// TwinCAT 3 PLC project virtual_plc
// ProgramVersion: 3.1.4024.0
// libraries:
//   Tc2_Standard, * (Beckhoff Automation GmbH)
//   Tc2_System, * (Beckhoff Automation GmbH)
//   Tc3_Module, * (Beckhoff Automation GmbH)
//   VisuSymbols,3.5.10.0,System
// project tree:
//   / Gestore di visualizzazione.TcVMO (not stored), GlobalTextList.TcGTLO, PlcTask.TcTTO
//   GVLs/ GVL.TcGVL
//   POUs/ LogMessage.TcPOU, MAIN.TcPOU, MaintenanceTask.TcPOU, status.TcDUT
//   VISU/ Visualization.TcVIS
// real-time tasks:
//   TASK PlcTask: cycle T#10ms, priority 20, ADS port 350

CONFIGURATION virtual_plc
    RESOURCE PLC ON TwinCAT3
        TASK PlcTask(INTERVAL := T#10ms, PRIORITY := 20);
        PROGRAM MAIN WITH PlcTask : MAIN;
    END_RESOURCE
END_CONFIGURATION

// ---- POUs/status.TcDUT
{attribute 'qualified_only'}
{attribute 'strict'}
TYPE status :
(START,
LEVELCHECK,
FILL,
HEAT,
HEATING,
BREW,
WATERREADY,
INTENSITY,
SUGAR,
READY,
CLEAN,
END,
OldState
) := START;
END_TYPE

// ---- GVLs/GVL.TcGVL
{attribute 'qualified_only'}
VAR_GLOBAL
	CoffeeReady: BOOL := FALSE;

	CLEANING: BOOL := FALSE;

	Message: STRING;
END_VAR

// ---- POUs/MAIN.TcPOU
PROGRAM MAIN

VAR
	start : BOOL := FALSE;
	Tfill: TON;
	FILLING : BOOL := FALSE;
	WaterLevel : BOOL := FALSE;
	Level : REAL;
	Theat: TON;
    WaterTemp :REAL;
	HEATING : BOOL := FALSE;
	Tbrew: TON;
    WaterReady : BOOL := FALSE;
	BREWING : BOOL := FALSE;
    Tend: TON;
	
	CoffeeBrewed : BOOL := FALSE;
	Tready: TON;
	
	INTENSITY_BUTTON : INT;
	TIMER : TON;
	SUGAR_BUTTON : INT :=1;
	SugarMessage : STRING(30);
	
	state : status := status.START;

	Tclean: TON;
END_VAR


CASE state OF

    status.START:  //initialization and start the machine
        GVL.CoffeeReady := FALSE; 
        FILLING := FALSE;
        HEATING := FALSE;
        BREWING := FALSE;
        WaterLevel := FALSE;
        WaterReady := FALSE;
		SugarMessage := '';
		LogMessage(msg := 'Machine started', cleaning := FALSE);
		IF start THEN
            state := status.LEVELCHECK; //check if the water is enough
        END_IF;       
	
    // over 80% is sufficient, otherwise the water has to be filled	
	status.LEVELCHECK: // over 80% is sufficient, otherwise the water has to be filled
	IF Level >= 80 THEN
		state := status.HEAT;
		WaterLevel := TRUE;
	ELSIF Level < 80 THEN
 		state:=status.FILL;
	END_IF
	
    //this status only if the water is under 80%
    status.FILL:  
		  Tfill(IN := TRUE, PT := T#8S);
		FILLING:= TRUE;
        FILLING := NOT WaterLevel; 
        WaterLevel := NOT FILLING;
        IF Tfill.Q THEN          
            Tfill(IN := FALSE);  
            FILLING := FALSE;    
            Level := 100;    
			LogMessage(msg := 'Water filled', cleaning := FALSE);
            State := status.HEAT;              
        END_IF
		IF NOT start THEN
			state := status.START;
		END_IF
		
	//when the water is checked, the heating process starts
	status.HEAT:
        Theat (IN:=TRUE, PT := T#5S);
		HEATING := TRUE;
		HEATING := NOT WaterReady;
		WaterReady := NOT HEATING;
		IF Theat.Q THEN
			HEATING := FALSE;
			WaterTemp := 100;
			Level := Level - 10;
			Theat(IN:= FALSE);
			state := status.WATERREADY;
		END_IF
		
	// when the right temperature of the water is reached, water is ready 
     status.WATERREADY:
	    WaterReady := TRUE;
        Theat(IN := TRUE, PT := T#5S);
        IF Theat.Q THEN
            WaterReady := FALSE;
            Theat(IN := FALSE);
			WaterTemp := 30;
            state := status.INTENSITY;
        END_IF
	// need to choose the intensity of the coffee, level 1 if the user wants light coffe and 3 if strong coffee
    status.INTENSITY:  
		 WaterLevel := FALSE;
         CASE INTENSITY_BUTTON OF
            1: Tbrew(IN := TRUE, PT := T#3S);
            2: Tbrew(IN := TRUE, PT := T#6S);
            3: Tbrew(IN := TRUE, PT := T#9S);
        ELSE
            Tbrew(IN := TRUE, PT := T#6S);  
        END_CASE
	
        BREWING := TRUE;  

        Tbrew (IN:=TRUE, PT:= T#5S);
        IF Tbrew.Q THEN
            BREWING := FALSE;     
            Tbrew(IN := FALSE); 
            State := status.SUGAR;  
            CoffeeBrewed := TRUE; 
        END_IF
		
	// the user can choose the sugar quantity
    status.SUGAR: 
		IF CoffeeBrewed := TRUE THEN
		CASE SUGAR_BUTTON OF
			1: SugarMessage := 'no sugar';
			2: SugarMessage := 'medium sugar';
			3: SugarMessage := 'full sugar';
		ELSE
            SugarMessage := 'invalid selection';
		END_CASE
		state := status.READY;
	END_IF
	
	//The coffee is ready
    status.READY:  
        Tready(IN := TRUE, PT := T#5S);
        IF Tready.Q THEN
            Tready(IN := FALSE);
            state := status.END;
            start := FALSE;
			GVL.CoffeeReady := TRUE;
			CoffeeBrewed := FALSE;
        END_IF
		
	
	status.END:  
        Tend(IN := TRUE, PT := T#5S);
        IF Tend.Q THEN           
            IF GVL.CLEANING THEN
				state:=status.CLEAN;
				Tend(IN := FALSE);
				start := FALSE;
				GVL.CoffeeReady := FALSE;
				
			ELSE 
            	Tend(IN := FALSE);
				start := FALSE;
				GVL.CoffeeReady := FALSE;
				state := status.START;
			END_IF
        END_IF;
		
	//waiting time to allow the machine cleaning program, if we reached 5 cycles
	status.CLEAN:
		 Tclean(IN:=TRUE, PT := T#8S);
		 IF Tclean.Q THEN
			 Tclean(IN:=FALSE);
			 state:=status.START;
			 
		 END_IF	  

END_CASE;

END_PROGRAM

// ---- POUs/LogMessage.TcPOU
FUNCTION LogMessage : BOOL
VAR_INPUT
	msg : STRING;
	cleaning :BOOL;
END_VAR
VAR
END_VAR

IF GVL.Message <> msg THEN
GVL.Message := msg;
END_IF;
GVL.CLEANING := cleaning;
LogMessage := TRUE;

END_FUNCTION

// ---- POUs/MaintenanceTask.TcPOU
PROGRAM MaintenanceTask
VAR
	CycleCounter: INT := 0;;
	MaintenanceNeeded: BOOL;
	Tclean: Ton;
	
	ResetCounter: BOOL;
	CoffeeReadyOld: BOOL := FALSE;
	
	bResult: BOOL;
	Treset: Ton;
END_VAR

// every cooffee made the counter increase
IF (GVL.CoffeeReady = TRUE) AND (CoffeeReadyOld = FALSE) THEN
    CycleCounter := CycleCounter + 1;
END_IF;

CoffeeReadyOld := GVL.CoffeeReady;

// if the machine has done 5 coffee, the cleaning part is needed
IF CycleCounter >= 5 THEN
    MaintenanceNeeded := TRUE;
   

    Tclean(IN := TRUE, PT := T#6S);
	LogMessage (msg := 'Maintenance required!', cleaning := TRUE);
    IF Tclean.Q THEN
        Tclean(IN := FALSE);
        ResetCounter := TRUE;
		LogMessage(msg := 'Maintenance done', cleaning := FALSE);
    END_IF;
//maintenance finished and numbur of coffe made
ELSE 
    MaintenanceNeeded := FALSE;
    LogMessage(msg := CONCAT('Coffees made: ', INT_TO_STRING(CycleCounter)), cleaning := FALSE);
	;
END_IF;

//after cleaning, counter must be resetted
IF ResetCounter = TRUE THEN  
    
LogMessage(msg := 'Maintenance done', cleaning := FALSE);
Treset(IN := TRUE, PT := T#2S);
    IF Treset.Q THEN
        Treset(IN := FALSE);
		CycleCounter := 0;
        ResetCounter := FALSE;
    END_IF;
END_IF;

END_PROGRAM

// ---- VISU/Visualization.TcVIS
VISUALIZATION Visualization  // 2x2
END_VISUALIZATION
